FUNCTION_BLOCK FB_TrajectoryGenerator
VAR_INPUT
END_VAR
VAR_OUTPUT
	fqPos : LREAL; //joint pos
	fqVel : LREAL; //joint vel
	fqAcc : LREAL; //joint acc
END_VAR
VAR
	fqStart : LREAL; //start pos
	fqFinal : LREAL; //goal ¨pos
	ftFinal : LREAL; //final time	
	

	a0  : LREAL := 0.0;
	a1  : LREAL := 0.0;
	a2  : LREAL := 0.0;
	a3  : LREAL := 0.0;
	a4  : LREAL := 0.0;
	a5  : LREAL := 0.0;
	
	
END_VAR

METHOD getTrajectory : BOOL
VAR_INPUT
	ftTraj : LREAL; // traj point
END_VAR

IF ftTraj <= ftFinal THEN
	fqPos := a0 + a1*EXPT(ftTraj,1) +  a2*EXPT(ftTraj,2) + a3*EXPT(ftTraj,3) + a4*EXPT(ftTraj,4) + a5*EXPT(ftTraj,5);
	fqVel := a1 +  2*a2*EXPT(ftTraj,1) + 3*a3*EXPT(ftTraj,2) + 4*a4*EXPT(ftTraj,3) + 5*a5*EXPT(ftTraj,4);
	fqAcc := 2*a2 + 2*3*a3*EXPT(ftTraj,1) + 3*4*a4*EXPT(ftTraj,2) + 4*5*a5*EXPT(ftTraj,3);
ELSE
	fqPos := fqFinal;
	fqVel := 0.0;
	fqAcc := 0.0;
END_IF
END_METHOD

METHOD init : BOOL
VAR_INPUT
	fqStartInit : LREAL; //start pos
	fqFinalInit : LREAL; //goal ¨pos
	ftFinalInit : LREAL; //final time	
END_VAR

fqStart := fqStartInit;
fqFinal := fqFinalInit;
ftFinal := ftFinalInit;

a0 := fqStartInit;
a1 := 0.0;
a2 := 0.0;
a3 := (10*(fqFinalInit - fqStartInit))/EXPT(ftFinalInit,3);
a4 := -(15*(fqFinalInit - fqStartInit))/EXPT(ftFinalInit,4);
a5 :=  (6*(fqFinalInit - fqStartInit))/EXPT(ftFinalInit,5);
END_METHOD

END_FUNCTION_BLOCK

(* stored: Version 1.1.0.1, ProductVersion 3.1.4024.9
   POU FB_TrajectoryGenerator: Id {377b08c1-e10b-45e1-9414-82eb9ae2dc7f}, SpecialFunc None
   Method getTrajectory: Id {cc7013b5-a934-4a59-ac2a-2227b2ae72a9}
   Method init: Id {d973b4a1-c418-4db1-97e2-1f7239ff7f26} *)
